KUKA KRL data list: $config.dat

&ACCESS RV$
&REL 1
DEFDAT $CONFIG
INT COM_ACTION=0
INT COM_ACTCNT=0
REAL COM_ROUNDM=0
REAL COM_VALUE1=0
REAL COM_VALUE2=0
REAL COM_VALUE3=0
REAL COM_VALUE4=0
DECL E6AXIS COM_E6AXIS
DECL POS COM_POS
DECL FRAME COM_FRAME
ENDDAT
